// TIA Portal project "E04_Antifurto_STEP_2" (V18)

(* hardware
DEVICE "S71500/ET200MP station_1"  S7-1500 station
   slot 0: "Telaio di montaggio_0"  Rack  6ES7 590-1***0-0AA0
   slot 1: "PLC_1"  CPU 1516-3 PN/DP  6ES7 516-3AN01-0AB0  V2.5
      slot 3: "Display CPU_1"  6ES7591-1BA00-0AA0
   slot 2: "DI 32x24VDC HF_1"  DI 32x24VDC HF  6ES7 521-1BL00-0AB0  V2.1
   slot 3: "DQ 32x24VDC/0.5A HF_1"  DQ 32x24VDC/0.5A HF  6ES7 522-1BL01-0AB0  V1.0
   slot 4: "AI 8xU/I/RTD/TC ST_1"  AI 8xU/I/RTD/TC ST  6ES7 531-7KF00-0AB0  V2.1
   slot 5: "AQ 4xU/I ST_1"  AQ 4xU/I ST  6ES7 532-5HD00-0AB0  V2.1
*)

// ===== PLC "PLC_1"  CPU 1516-3 PN/DP =====

VAR_GLOBAL   // PLC tag table "Tabella delle variabili standard"
   "led00" AT %Q0.0 : Bool;
   "led01" AT %Q0.1 : Bool;
   "led02" AT %Q0.2 : Bool;
   "led03" AT %Q0.3 : Bool;
   "led04" AT %Q0.4 : Bool;
   "led05" AT %Q0.5 : Bool;
   "led06" AT %Q0.6 : Bool;
   "led07" AT %Q0.7 : Bool;
   "led10" AT %Q1.0 : Bool;
   "led11" AT %Q1.1 : Bool;
   "led12" AT %Q1.2 : Bool;
   "led13" AT %Q1.3 : Bool;
   "led14" AT %Q1.4 : Bool;
   "led15" AT %Q1.5 : Bool;
   "led16" AT %Q1.6 : Bool;
   "led17" AT %Q1.7 : Bool;
   "led20" AT %Q2.0 : Bool;
   "led21" AT %Q2.1 : Bool;
   "led22" AT %Q2.2 : Bool;
   "led23" AT %Q2.3 : Bool;
   "led24" AT %Q2.4 : Bool;
   "led25" AT %Q2.5 : Bool;
   "led26" AT %Q2.6 : Bool;
   "led27" AT %Q2.7 : Bool;
   "LA" AT %Q3.0 : Bool;
   "led31" AT %Q3.1 : Bool;
   "led32" AT %Q3.2 : Bool;
   "led33" AT %Q3.3 : Bool;
   "led34" AT %Q3.4 : Bool;
   "led35" AT %Q3.5 : Bool;
   "led36" AT %Q3.6 : Bool;
   "led37" AT %Q3.7 : Bool;
END_VAR

DATA_BLOCK "DB_Comandi"   // DB1
{ S7_Optimized_Access := 'TRUE' }
VERSION : 0.1
   VAR
      btnStop : Bool;
      btnAuto : Bool;
      btnMan : Bool;
      btnReset : Bool;
      btnEmergenza : Bool;
   END_VAR
BEGIN
END_DATA_BLOCK

DATA_BLOCK "DB_Stati"   // DB2
{ S7_Optimized_Access := 'TRUE' }
VERSION : 0.1
   VAR
      sAuto : Bool;
      sStop : Bool;
      sMan : Bool;
      sHome : Bool;
      sAttesaStop : Bool;
      sEmergenza : Bool;
      blni1 : Bool;
      bRip1 : Bool;
   END_VAR
BEGIN
END_DATA_BLOCK

DATA_BLOCK "DB_Tappe"   // DB3
{ S7_Optimized_Access := 'TRUE' }
VERSION : 0.1
   VAR
      tappeGemma : Int;
      tappeM1 : Int;
   END_VAR
BEGIN
END_DATA_BLOCK

DATA_BLOCK "DB_Variabili"   // DB4
{ S7_Optimized_Access := 'TRUE' }
VERSION : 0.1
   VAR
      timerResetPulsantiSTART : Bool;
      timerResetPulsantiDONE : Bool;
      timerResetPulsantiOUTPUT : Time;
      timerResetPulsantiDURATA : Time;
      cont : Int;
      i : Int;
      P : Bool;
      F1 : Bool;
      F2 : Bool;
      LA : Bool;
      "M" : Bool;
   END_VAR
BEGIN
END_DATA_BLOCK

// folder: System blocks/Program resources

DATA_BLOCK "timerResetPulsanti"   // DB5
{ S7_Optimized_Access := 'TRUE' }
AUTHOR : Simatic
FAMILY : IEC
NAME : IEC_TMR
VERSION : 1.0
// stored: InstanceOfName IEC_TIMER
"IEC_TIMER"
BEGIN
END_DATA_BLOCK

// folder: (top level)

FUNCTION "FC_Gemma" : Void   // FC1, SCL
{ S7_Optimized_Access := 'TRUE' }
VERSION : 0.1
BEGIN
   CASE "DB_Tappe".tappeGemma OF
       0: //Stato di Riposo
           "DB_Stati".sStop := TRUE;
           IF "DB_Comandi".btnAuto = TRUE THEN
               "DB_Tappe".tappeGemma := 1; //Home
               "DB_Stati".sAttesaStop := FALSE;
               "DB_Stati".sAuto := FALSE;
               "DB_Stati".sHome := TRUE;
               "DB_Stati".sMan := FALSE;
               "DB_Stati".sStop := FALSE;
               "DB_Stati".sEmergenza := FALSE;
           ELSE
               IF "DB_Comandi".btnMan = TRUE THEN
                   "DB_Tappe".tappeGemma := 4; //Manuale
                   "DB_Stati".sAttesaStop := FALSE;
                   "DB_Stati".sAuto := FALSE;
                   "DB_Stati".sHome := FALSE;
                   "DB_Stati".sMan := TRUE;
                   "DB_Stati".sStop := FALSE;
                   "DB_Stati".sEmergenza := FALSE;
               END_IF;
           END_IF;

        1: //Stato di Home
            IF "DB_Stati".blni1 = TRUE  THEN
                "DB_Tappe".tappeGemma := 2; //Automatico
                "DB_Stati".sAttesaStop := FALSE;
                "DB_Stati".sAuto := TRUE;
                "DB_Stati".sHome := FALSE;
                "DB_Stati".sMan := FALSE;
                "DB_Stati".sStop := FALSE;
                "DB_Stati".sEmergenza := FALSE;
            END_IF;

        2: //Stato di Automatico
            IF "DB_Comandi".btnStop = TRUE THEN
                "DB_Tappe".tappeGemma := 3; //Attesa Stop
                "DB_Stati".sAttesaStop := TRUE;
                "DB_Stati".sAuto := FALSE;
                "DB_Stati".sHome := FALSE;
                "DB_Stati".sMan := FALSE;
                "DB_Stati".sStop := FALSE;
                "DB_Stati".sEmergenza := FALSE;
            END_IF;

        3: //Stato di Attesa Stop
            IF "DB_Stati".bRip1 = TRUE THEN
                "DB_Tappe".tappeGemma := 0; //Stop
                "DB_Stati".sAttesaStop := FALSE;
                "DB_Stati".sAuto := FALSE;
                "DB_Stati".sHome := FALSE;
                "DB_Stati".sMan := FALSE;
                "DB_Stati".sStop := TRUE;
                "DB_Stati".sEmergenza := FALSE;
            END_IF;

        4: //Stato di Manuale
            IF "DB_Comandi".btnStop = TRUE THEN
                "DB_Tappe".tappeGemma := 0; //Stop
                "DB_Stati".sAttesaStop := FALSE;
                "DB_Stati".sAuto := FALSE;
                "DB_Stati".sHome := FALSE;
                "DB_Stati".sMan := FALSE;
                "DB_Stati".sStop := TRUE;
                "DB_Stati".sEmergenza := FALSE;
            END_IF;

        5: //Stato di Emergenza
            IF "DB_Comandi".btnEmergenza = TRUE AND "DB_Stati".sEmergenza THEN
                "DB_Tappe".tappeGemma := 0; //Stop
                "DB_Stati".sAttesaStop := FALSE;
                "DB_Stati".sAuto := FALSE;
                "DB_Stati".sHome := FALSE;
                "DB_Stati".sMan := FALSE;
                "DB_Stati".sStop := TRUE;
                "DB_Stati".sEmergenza := FALSE;
            END_IF;
    END_CASE;

    //Gestione Emergenza
    //
    IF "DB_Comandi".btnEmergenza = FALSE THEN
        "DB_Tappe".tappeGemma := 5; //Emergenza
        "DB_Stati".sAttesaStop := FALSE;
        "DB_Stati".sAuto := FALSE;
        "DB_Stati".sHome := FALSE;
        "DB_Stati".sMan := FALSE;
        "DB_Stati".sStop := FALSE;
        "DB_Stati".sEmergenza := TRUE;
    END_IF;
END_FUNCTION

FUNCTION "FC_Grafcet" : Void   // FC2, SCL
{ S7_Optimized_Access := 'TRUE' }
VERSION : 0.1
BEGIN
   //Imposto bIni e bRip a TRUE. Andranno poi gestiti in base alle condizioni dell'impianto
   //
   "DB_Stati".blni1 := TRUE;
   "DB_Stati".bRip1 := TRUE;

   //Gestisco il reset
   //
   IF "DB_Comandi".btnReset = TRUE AND "DB_Stati".sStop = TRUE THEN
      //reimposto le condizioni iniziali solo se la macchina è in stop
      //
       "DB_Tappe".tappeGemma := 0;
       "DB_Tappe".tappeM1 := 0;
   END_IF;

   //Gestisco il grafcet in questo caso il gioco di luci
   //

   //se P=TRUE e F1=TRUE
   //se P=FALSE e (F1=TRUE e F2=TRUE)
   //se P=TRUE e F1=TRUE e F2=TRUE
   //
   //Aggiungere Attiva (bStart) e Disattiva (bStop) antifurto
   //Aggiungere totale (bAuto) e Parziale (bMan)
   //Aggiungere sensore movimento M che vale TRUE se qualcosa si muove nella stanza
   //se M=TRUE allora LA=TRUE
   //In funzionamento parziale il sensore M viene ignorato
   //
   //ATTENZIONE in un programma PLC devo avere un unico punto in cui imposto un'uscita a TRUE o FALSE
   //
   IF "DB_Stati".sStop = TRUE THEN
       "DB_Variabili".LA := FALSE;
   END_IF;

   IF "DB_Stati".sAuto = TRUE THEN
       IF (("DB_Variabili".P = TRUE AND "DB_Variabili".F1 = TRUE) OR
           ("DB_Variabili".P = FALSE AND ("DB_Variabili".F1 = TRUE AND "DB_Variabili".F2 = TRUE)) OR
           ("DB_Variabili".P = TRUE AND ("DB_Variabili".F1 = TRUE AND "DB_Variabili".F2 = TRUE))) OR
           ("DB_Variabili".M = TRUE) THEN
           "DB_Variabili".LA := TRUE;
       ELSE
           "DB_Variabili".LA := FALSE;
       END_IF;

   END_IF;

   IF "DB_Stati".sMan = TRUE THEN
       IF ("DB_Variabili".P = TRUE AND "DB_Variabili".F1 = TRUE) OR
           ("DB_Variabili".P = FALSE AND ("DB_Variabili".F1 = TRUE AND "DB_Variabili".F2 = TRUE)) OR
           ("DB_Variabili".P = TRUE AND ("DB_Variabili".F1 = TRUE AND "DB_Variabili".F2 = TRUE)) THEN
           "DB_Variabili".LA := TRUE;
       ELSE
           "DB_Variabili".LA := FALSE;
       END_IF;
   END_IF;
END_FUNCTION

FUNCTION "FC_ResetPulsanti" : Void   // FC3, SCL
{ S7_Optimized_Access := 'TRUE' }
VERSION : 0.1
BEGIN
   IF "DB_Comandi".btnAuto = TRUE OR
       "DB_Comandi".btnMan = TRUE OR
       "DB_Comandi".btnReset = TRUE OR
       "DB_Comandi".btnStop = TRUE THEN
       "DB_Variabili".timerResetPulsantiSTART := TRUE;
   END_IF;

   IF "DB_Variabili".timerResetPulsantiDONE = TRUE THEN
       "DB_Variabili".timerResetPulsantiSTART := FALSE;
       "DB_Variabili".timerResetPulsantiDONE := FALSE;
       "DB_Comandi".btnAuto := FALSE;
       "DB_Comandi".btnMan := FALSE;
       "DB_Comandi".btnReset := FALSE;
       "DB_Comandi".btnStop := FALSE;
   END_IF;
END_FUNCTION

FUNCTION "FC_Timer" : Void   // FC4, SCL
{ S7_Optimized_Access := 'TRUE' }
VERSION : 0.1
BEGIN
   "DB_Variabili".timerResetPulsantiDURATA := T#500ms;

   "timerResetPulsanti".TON(IN:="DB_Variabili".timerResetPulsantiSTART,
                            PT:="DB_Variabili".timerResetPulsantiDURATA,
                            Q=>"DB_Variabili".timerResetPulsantiDONE,
                            ET=>"DB_Variabili".timerResetPulsantiOUTPUT);

   //
END_FUNCTION

FUNCTION "FC_Uscite" : Void   // FC5, SCL
{ S7_Optimized_Access := 'TRUE' }
VERSION : 0.1
BEGIN
   //Prima di scrivere fisicamente le uscite devo controllae che tutte le condizioni siano rispettate:
   //emergenza, protezioni fotucellula ecc...
   //
   "LA" := "DB_Variabili".LA;
END_FUNCTION

ORGANIZATION_BLOCK "Main"   // OB1, LAD, ProgramCycle
TITLE = "Main Program Sweep (Cycle)"
{ S7_Optimized_Access := 'TRUE' }
VERSION : 0.1
   VAR_INPUT
      Initial_Call : Bool;   // Initial call of this OB
      Remanence : Bool;   // =True, if remanent data are available
   END_VAR
   VAR_TEMP   // added for the SCL form of the ladder/FBD networks
      _w1 : Bool;
      _w2 : Bool;
      _w3 : Bool;
      _w4 : Bool;
   END_VAR
BEGIN

REGION Network 1
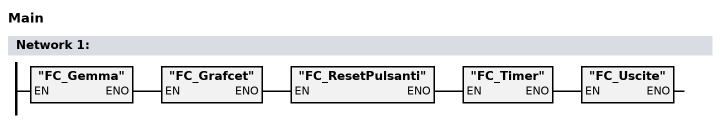
   RUNG wire#powerrail
      "FC_Gemma"()
      "FC_Grafcet"()
      "FC_ResetPulsanti"()
      "FC_Timer"()
      "FC_Uscite"()
   END_RUNG
   // the same network as SCL:
   "FC_Gemma"(ENO => #_w1);
   "FC_Grafcet"(EN := #_w1, ENO => #_w2);
   "FC_ResetPulsanti"(EN := #_w2, ENO => #_w3);
   "FC_Timer"(EN := #_w3, ENO => #_w4);
   IF #_w4 THEN "FC_Uscite"(); END_IF;
END_REGION
END_ORGANIZATION_BLOCK